(* IEC 61131-3 sources: ics/BLR101_ProenixContact/BLR101_1_ILC171_44/LogicalPOUs/Burner, 2 files *)

(* ---- BurnerFB.ST ---- *)
(*@PROPERTIES_EX@
TYPE: POU
LOCALE: 0
IEC_LANGUAGE: ST
PLC_TYPE: independent
PROC_TYPE: independent
GROUP: Burner
*)
(*@KEY@:DESCRIPTION*)

(*@KEY@:END_DESCRIPTION*)
FUNCTION_BLOCK BurnerFB

(*Group:Default*)

VAR
    TON_Overtime :	TON;
END_VAR

VAR_IN_OUT
    Brn_strct :	Brnr;
END_VAR

VAR
    AlarmFeedback :	BOOL;
    RunManual :	BOOL;
    RunAuto :	BOOL;
    COM :	BOOL;
    EnableMotorAuto :	BOOL;
END_VAR

VAR_INPUT
    Cycle :	Cycle;
    SetOvertime :	TIME;
END_VAR

VAR
    AlarmBlock :	BOOL;
END_VAR

(*@KEY@: WORKSHEET
NAME: BurnerFB
IEC_LANGUAGE: ST
*)
    (*Alarm Feedback processing*)
TON_Overtime(IN:=Brn_strct.CW.Enable and
    ((Brn_strct.SW.COM and not Brn_strct.SW.RUN) or
    (not Brn_strct.SW.COM and Brn_strct.SW.RUN)),PT:=SetOvertime);

if TON_Overtime.Q then
    AlarmFeedback:=true;
end_if;
if not Brn_strct.CW.ExtraEn and Brn_strct.SW.COM then
    AlarmBlock:= true;
end_if;

if AlarmFeedback or Brn_strct.CW.ExtraAlarm or AlarmBlock then
    Brn_strct.SW.AlarmAccum:= true;
end_if;

if Brn_strct.CW.ACK then
    AlarmFeedback:=false;
    AlarmBlock:= false;
    Brn_strct.SW.AlarmAccum:= false;
end_if;

    (*Auto/Manual mode selection*)
if Brn_strct.CW.EnableAuto then
    Brn_strct.SW.Auto:= true;
elsif Brn_strct.CW.DisableAuto then
    Brn_strct.SW.Auto:= false;
end_if;

Brn_strct.SW.ManOK:= not Brn_strct.SW.AlarmAccum and Brn_strct.CW.AuxON and
    Brn_strct.CW.Enable and not Brn_strct.SW.Auto;

Brn_strct.SW.AutoOK:= not Brn_strct.SW.AlarmAccum and Brn_strct.CW.AuxON and
    Brn_strct.CW.Enable and Brn_strct.SW.Auto and Cycle.SW.Running;

    (*Manual mode activation*)
if Brn_strct.CW.ManStart then
    RunManual:=true;
end_if;
if Brn_strct.CW.ManStop or not Brn_strct.SW.ManOK then
    RunManual:=false;
end_if;

    (*Auto mode activation*)
RunAuto:= (Cycle.CW.PulseStart or RunAuto) and Brn_strct.SW.AutoOK and
    Brn_strct.SW.Auto;

    (*Set command for start*)
COM:=((RunManual and Brn_strct.SW.ManOK) or (RunAuto and Brn_strct.SW.AutoOK and
    Brn_strct.CW.AutoON));

Brn_strct.SW.COM:=COM and not Brn_strct.CW.SimEn;

    (*SP limatation*)
if Brn_strct.Sys.MaxSP > 100.0 then
    Brn_strct.Sys.MaxSP:=100.0;
elsif Brn_strct.Sys.MaxSP < 0.0 then
    Brn_strct.Sys.MaxSP:=0.0;
end_if;

if Brn_strct.Sys.MinSP > 100.0 then
    Brn_strct.Sys.MinSP:=100.0;
elsif Brn_strct.Sys.MinSP < 0.0 then
    Brn_strct.Sys.MinSP:=0.0;
end_if;

if Brn_strct.Sys.MinSP > Brn_strct.Sys.MaxSP then
    Brn_strct.Sys.MinSP:=Brn_strct.Sys.MaxSP;
end_if;

if Brn_strct.Sys.ManSP > Brn_strct.Sys.MaxSP then
    Brn_strct.Sys.ManSP:=Brn_strct.Sys.MaxSP;
elsif Brn_strct.Sys.ManSP < Brn_strct.Sys.MinSP then
    Brn_strct.Sys.ManSP:=Brn_strct.Sys.MinSP;
end_if;

if Brn_strct.Sys.AutoSP > Brn_strct.Sys.MaxSP then
    Brn_strct.Sys.AutoSP:=Brn_strct.Sys.MaxSP;
elsif Brn_strct.Sys.AutoSP < Brn_strct.Sys.MinSP then
    Brn_strct.Sys.AutoSP:=Brn_strct.Sys.MinSP;
end_if;

    (*Status processing*)
if Brn_strct.SW.AlarmAccum then                                                 (*Alarm*)
    Brn_strct.Sys.Status:=word#2;
elsif not Brn_strct.CW.ExtraEn then                                             (*Blocking*)
    Brn_strct.Sys.Status:=word#4;
elsif Brn_strct.SW.COM then                                                     (*Working*)
    Brn_strct.Sys.Status:=word#1;
else                                                                            (*Stoped*)
    Brn_strct.Sys.Status:=word#0;
end_if;

Brn_strct.CW.EnableAuto:=false;
Brn_strct.CW.DisableAuto:=false;
Brn_strct.CW.ManStart:=false;
Brn_strct.CW.ManStop:=false;
Brn_strct.CW.ACK:=false;
(*@KEY@: END_WORKSHEET *)
END_FUNCTION_BLOCK

(* ---- Burner_section.ST ---- *)
(*@PROPERTIES_EX@
TYPE: POU
LOCALE: 0
IEC_LANGUAGE: ST
PLC_TYPE: independent
PROC_TYPE: independent
GROUP: Burner
*)
(*@KEY@:DESCRIPTION*)

(*@KEY@:END_DESCRIPTION*)
PROGRAM Burner_section

(*Group:Default*)

VAR
    Burner :	BurnerFB;
END_VAR

VAR_EXTERNAL
    Boiler :	Blr;
    Cycle :	Cycle;
    xBrnRemote :	BOOL;
    xBrnQM_ON :	BOOL;
    xBrnSafetyCircON :	BOOL;
    xBrnRUN :	BOOL;
    xBrnFault :	BOOL;
    xBrnUnlock :	BOOL;
    xBrnCOM :	BOOL;
    arrMB_Srv1Data :	MB2_TCP_ARR_W_0_7167;
END_VAR

VAR
    BrnPID :	BACL_PID_T1_V0_10;
END_VAR

VAR_EXTERNAL
    BrnrSP :	REAL;
    BrnrFeedback :	Snsr;
    arrSlvReadData :	SlvReadData;
END_VAR

VAR
    rBrnPidDeviation :	REAL;
END_VAR

VAR_EXTERNAL
    TestFlag :	BOOL;
END_VAR

(*@KEY@: WORKSHEET
NAME: Burner_section
IEC_LANGUAGE: ST
*)
    (*Burner DI*)
Boiler.Brn1.CW.Enable:= xBrnRemote;
Boiler.Brn1.CW.AuxON:= Cycle.CW.AuxON;
Boiler.Brn1.CW.ExtraEn:= xBrnSafetyCircON and xBrnQM_ON;
Boiler.Brn1.CW.ExtraAlarm:= xBrnFault;
Boiler.Brn1.SW.Rem:= xBrnRemote;
Boiler.Brn1.SW.RUN:= xBrnRUN or (Boiler.Brn1.Sys.Phase > word#12);

    (*Burner FB call*)
Burner(Brn_strct:=Boiler.Brn1,Cycle:=Cycle,SetOvertime:=t#90s);
Boiler.Brn1:=Burner.Brn_strct;
    (*ModBusArray ControlWord Reset*)
arrMB_Srv1Data[100]:=word#0;

    (*Burner D0*)
xBrnUnlock:= Boiler.Brn1.CW.ACK;
xBrnCOM:= Boiler.Brn1.SW.COM;

    (*Burning controller parameters*)
Boiler.Brn1.Sys.Phase:= arrSlvReadData[0][1];
Boiler.Brn1.Sys.CurrOut:= real_to_word(BrnrFeedback.RealValue)(*arrSL1_ReadData[0][11]*);
Boiler.Brn1.Sys.CurrSP:= arrSlvReadData[0][12];
Boiler.Brn1.Sys.CurrPV:= arrSlvReadData[0][13];
Boiler.Brn1.Sys.FlameVal:= (arrSlvReadData[0][14] / word#10);
Boiler.Brn1.SW.FireOK:= (Boiler.Brn1.Sys.FlameVal > word#0);

Boiler.Brn1.Sys.StartUpCount.W0:= arrSlvReadData[4][22];
Boiler.Brn1.Sys.StartUpCount.W1:= arrSlvReadData[4][23];
Boiler.Brn1.Sys.HoursCount.W0:= arrSlvReadData[4][24];
Boiler.Brn1.Sys.HoursCount.W1:= arrSlvReadData[4][25];

Boiler.Brn1.Sys.ErrCode:= arrSlvReadData[4][26];
Boiler.Brn1.Sys.DiagCode:= arrSlvReadData[4][27];
Boiler.Brn1.Sys.ErrClass:= arrSlvReadData[4][28];

    (*Burner PID*)
BrnPID(IN_xEnable:=Boiler.Brn1.Reg[0].CW.En,
    IN_tCycleTime:=t#500ms,
    IN_rSetPoint:=Boiler.Brn1.Reg[0].SP,
    IN_rActValue:=Boiler.AI[1].RealValue,
    IN_rDeadBand:=Boiler.Brn1.Reg[0].DeadBand,
    IN_rYmax:=(Boiler.Brn1.Sys.MaxSP * 10.0),
    IN_rYmin:=(Boiler.Brn1.Sys.MinSP * 10.0),
    IN_rYoff:=Boiler.Brn1.Reg[0].ManVal,
    IN_rKR:=Boiler.Brn1.Reg[0].Kp,
    IN_rTN:=Boiler.Brn1.Reg[0].Tn,
    IN_rTV:=Boiler.Brn1.Reg[0].Tv);

Boiler.Brn1.Reg[0].Y:=BrnPID.OUT_rYout;
rBrnPidDeviation:=BrnPID.OUT_rControlDeviation;

if Boiler.Brn1.SW.Auto then
    BrnrSP:= Boiler.Brn1.Sys.AutoSP;
else
    BrnrSP:= Boiler.Brn1.Sys.ManSP;
end_if;

(*@KEY@: END_WORKSHEET *)
END_PROGRAM
